// TIA Portal V17 export
// export: Created 2024-09-02T12:50:33.5991001Z, ExportSetting WithDefaults, DisplayName Totally Integrated Automation Portal, DisplayVersion V17, DisplayName TIA Portal Openness, DisplayVersion V17, DisplayName TIA Portal Version Control Interface, DisplayVersion V17, DisplayName STEP 7 Professional, DisplayVersion V17, DisplayName STEP 7 Safety, DisplayVersion V17, DisplayName WinCC Professional, DisplayVersion V17
TYPE "TypeMobySequenz"
// stored: IsFailsafeCompliant false
   STRUCT
      WorkArea : Struct   // Auftragsfach / Job mailbox
         SequenceNr : Int;   // aktuelle Sequenznummer / current sequence number
         Function : Int;   // 1= Lesen; 2= Schreiben / 1= Read; 2= Write
         ADDR_TAG : Int;   // Adresse auf dem MDS / Address on the MDS
         LEN_DATA : Int;   // Anzahl Byte für Auftrag / Number of bytes for job
      END_STRUCT;
      Results : Struct   // Ergebnisfach / Result compartment
         SequenceNr : Int;   // aktuelle Sequenznummer / current sequence number
         Function : Int;   // 1= Lesen; 2= Schreiben / 1= Read; 2= Write
         ReadyForOrder : Bool;   // ASM Bereit für Auftrag / ASM Ready for order
      END_STRUCT;
   END_STRUCT;
END_TYPE
